(* PLC project Unnamed, Unknown Unnamed 1 *)
(* stored: creationDateTime 2024-12-02T17:14:16, modificationDateTime 2024-12-02T17:21:52 *)

PROGRAM exp2
  VAR_INPUT
    Start : BOOL;
    Stop : BOOL;
  END_VAR
  VAR_OUTPUT
    Motor : BOOL;
  END_VAR

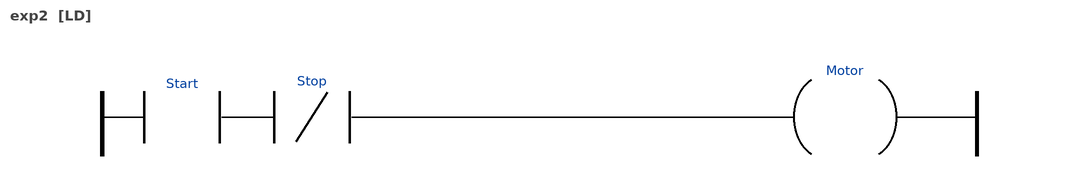
(* LD diagram, written out as Structured Text *)
Motor := Start AND NOT Stop;
END_PROGRAM

CONFIGURATION Config0
  RESOURCE Res0 ON PLC
    TASK task0(INTERVAL := T#20ms, PRIORITY := 0);
    PROGRAM instance0 WITH task0 : exp2;
  END_RESOURCE
END_CONFIGURATION
